INTERFACE I_Magnetventil

METHOD M_M_OEFFNEN : BOOL
VAR_INPUT
END_VAR
END_METHOD

METHOD M_M_SCHLIESSEN : BOOL
VAR_INPUT
END_VAR
END_METHOD

END_INTERFACE

(* stored: Version 1.1.0.1, ProductVersion 3.1.4024.12
   Itf I_Magnetventil: Id {a17bf922-bf26-4dd4-85a2-f2356bfb708a}
   Method M_M_OEFFNEN: Id {bc3072cc-c19f-4ad0-a0a3-0b54b2223672}
   Method M_M_SCHLIESSEN: Id {ccf9c1a0-1761-4444-8cdc-e453baac0299} *)
